Staubli VAL3: Txt_initData.pgx

program Txt_initData()
  local num l_nInit
begin
  //    title("Please Enter Txt Files Total number")
  //  cls()
  //  popUpMsg("请在点击OK后输入txt文档总包数（显示在左下角），并点回车。如需修改，选择F7重新进行初始化")
  //  get(nTxtTotal)
  //  putln(nTxtTotal)
  //  call Txt_initData()
  while size(sString)>1
    $ddel(sString,size(sString)-1)
  endWhile
  while size(nPulse)>1
    $ddel(nPulse,size(nPulse)-1)
  endWhile
  while size(pfrmCad)>1
    $ddel(pfrmCad,size(pfrmCad)-1)
  endWhile
  pfrmCad[0].trsf={0,0,0,0,0,0}
  sString[0]=""
  for l_nInit=1 to 1499
    $dins(sString,l_nInit)
    $dins(nPulse,l_nInit)
    $dins(pfrmCad,l_nInit)
  endFor
  bTxtPrSv=false
  //  popUpMsg("txt is ready")
end
